Staubli VAL3: pub.pjx

--- pub.pjx ---
Parameters version=s7.8.3 stackSize=5000 millimeterUnit=true
Program file=main.pgx
Program file=stop.pgx
Data file=pub.dtx

--- main.pgx ---
public program main()
begin
end
